// TwinCAT 3 PLC project PLC1
// ProgramVersion: 3.1.4023.0
// libraries:
//   CmpBitmapPool, * (System)
//   Tc2_MC2, * (Beckhoff Automation GmbH)
//   Tc2_Standard, * (Beckhoff Automation GmbH)
//   Tc2_System, * (Beckhoff Automation GmbH)
//   Tc3_Module, * (Beckhoff Automation GmbH)
//   VisuDialogs, * (System)
//   VisuSymbols,3.5.10.0,System
// project tree:
//   / GlobalTextList.TcGTLO (not stored), ImagePool.TcIPO (not stored), PlcTask.TcTTO, Visualization Manager.TcVMO (not stored)
//   GVLs/ GVL.TcGVL
//   POUs/ blinker.TcPOU (not stored), control.TcPOU, light.TcPOU, MAIN.TcPOU (not stored), motor.TcPOU
//   VISUs/ Huoltosivu.TcVIS (not stored), Visualization.TcVIS
// real-time tasks:
//   TASK PlcTask: cycle T#10ms, priority 20, ADS port 350
// motion (NC):
//   TASK NC-Task 1 SAF: cycle T#2ms, priority 4, ADS port 501
//   TASK NC-Task 1 SVB: cycle T#10ms, priority 8, ADS port 511
//   AXIS Axis 1, stepper (id 1)
//     Velo: Maximum=942.478
//     OtherSettings: AllowMotionCmdToSlave=true
//     encoder EncType=4
//       EncPara: ScaleFactorNumerator=0.007363107781851, MaxCount=#x0000ffff
//         Inc: RefSearchInverse=true, RefSyncInverse=false, RefMode=1, RefSoftSyncMask=#x0000ffff
//         TimeComp: TimeCompMode=1, EncDelayCycles=4
//     drive DrvType=24
//       Analog: VeloReferenz=942.477796076938, TorqueSetpointScale=10, ScaleFactorActTorque=0.1
//       TimeComp: TaskDelayCycles=1
//     controller CtrType=1
//       CtrPara: PriorControlFactor=1
//         Observer: BandWidth=20
//   AXIS Axis 2, servo (id 2)
//     OtherSettings: AllowMotionCmdToSlave=true
//     encoder EncType=19
//       EncPara: MaxCount=#xffffffff
//     drive DrvType=16
//       DrvPara: MaxCount=#xffffffff, DriveControlDWord=#x00020000
//         Analog: TorqueSetpointScale=10, ScaleFactorActTorque=0.1
//         TimeComp: TaskDelayCycles=1
//     controller CtrType=1
//       CtrPara: PriorControlFactor=1
//         Observer: BandWidth=20
// I/O:
//   DEVICE Device 1 (EtherCAT), AmsNetId 192.168.0.5.2.1
//     Term 1 (EK1200) [EK1200-5000 EtherCAT Power supply (2A E-Bus)]
//       Term 2 (EL1004) [EL1004 4Ch. Dig. Input 24V, 3ms]
//       Term 3 (EL1008) [EL1008 8Ch. Dig. Input 24V, 3ms]
//       Term 4 (EL2004) [EL2004 4Ch. Dig. Output 24V, 0.5A]
//       Term 5 (EL2008) [EL2008 8Ch. Dig. Output 24V, 0.5A]
//       Term 6 (EL3102) [EL3102 2Ch. Ana. Input +/-10V, Diff.]
//       Term 7 (EL4132) [EL4132 2Ch. Ana. Output +/-10V, 16bit]
//       Term 8 (EK1110) [EK1110 EtherCAT extension]
//     Term 9 (EK1100) [EK1100 EtherCAT Coupler (2A E-Bus)]
//       Term 10 (EL7031) [EL7031 1Ch. Stepper motor output stage (24V, 1.5A)]
//       Term 11 (EL7211-0010) [EL7211-0010 1Ch. MDP742 Servo motor output stage with OCT (50V, 4.5A RMS)]
//       Term 12 (EL9011) [EL9011 End Terminal]
//   DEVICE Device 5 (COM Port)
// variable links:
//   NC-Task 1 SAF/Axes/Axis 1, stepper <-> Device 1 (EtherCAT)/Term 9 (EK1100)/Term 10 (EL7031)
//     Drive/Inputs/In/nState1 @bit 3 <-> STM Status/Status/Error
//     Drive/Inputs/In/nState1 @bit 5 <-> STM Status/Status/Moving negative
//     Drive/Inputs/In/nState1 @bit 4 <-> STM Status/Status/Moving positive
//     Drive/Inputs/In/nState1 @bit 1 <-> STM Status/Status/Ready
//     Drive/Inputs/In/nState1 <-> STM Status/Status/Ready to enable
//     Drive/Inputs/In/nState1 @bit 6 <-> STM Status/Status/Torque reduced
//     Drive/Inputs/In/nState1 @bit 2 <-> STM Status/Status/Warning
//     Drive/Inputs/In/nState2 @bit 3 <-> STM Status/Status/Digital input 1
//     Drive/Inputs/In/nState2 @bit 4 <-> STM Status/Status/Digital input 2
//     Drive/Inputs/In/nState2 @bit 5 <-> STM Status/Status/Sync error
//     Drive/Inputs/In/nState2 @bit 7 <-> STM Status/Status/TxPDO Toggle
//     Drive/Inputs/In/nState4 @bit 1 <-> WcState/InputToggle
//     Drive/Inputs/In/nState4 <-> WcState/WcState
//     Drive/Outputs/Out/nCtrl1 <-> STM Control/Control/Enable
//     Drive/Outputs/Out/nCtrl1 @bit 2 <-> STM Control/Control/Reduce torque
//     Drive/Outputs/Out/nCtrl1 @bit 1 <-> STM Control/Control/Reset
//     Drive/Outputs/Out/nDataOut2[0] <-> STM Velocity/Velocity
//     Enc/Inputs/In/nDataIn1[0] <-> ENC Status compact/Counter value
//     Enc/Inputs/In/nDataIn2[0] <-> ENC Status compact/Latch value
//     Enc/Inputs/In/nState1 @bit 4 <-> ENC Status compact/Status/Counter overflow
//     Enc/Inputs/In/nState1 @bit 3 <-> ENC Status compact/Status/Counter underflow
//     Enc/Inputs/In/nState1 @bit 1 <-> ENC Status compact/Status/Latch extern valid
//     Enc/Inputs/In/nState1 @bit 2 <-> ENC Status compact/Status/Set counter done
//     Enc/Inputs/In/nState2 @bit 4 <-> ENC Status compact/Status/Status of extern latch
//     Enc/Inputs/In/nState2 @bit 5 <-> ENC Status compact/Status/Sync error
//     Enc/Inputs/In/nState2 @bit 7 <-> ENC Status compact/Status/TxPDO Toggle
//     Enc/Inputs/In/nState4 @bit 1 <-> WcState/InputToggle
//     Enc/Inputs/In/nState4 <-> WcState/WcState
//     Enc/Outputs/Out/nCtrl1 @bit 3 <-> ENC Control compact/Control/Enable latch extern on negative edge
//     Enc/Outputs/Out/nCtrl1 @bit 1 <-> ENC Control compact/Control/Enable latch extern on positive edge
//     Enc/Outputs/Out/nCtrl1 @bit 2 <-> ENC Control compact/Control/Set counter
//     Enc/Outputs/Out/nDataOut1[0] <-> ENC Control compact/Set counter value
//   NC-Task 1 SAF/Axes/Axis 2, servo <-> Device 1 (EtherCAT)/Term 9 (EK1100)/Term 11 (EL7211-0010)
//     Drive/Inputs/In/nDcOutputTime <-> InfoData/DcOutputShift
//     Drive/Inputs/In/nState1 <-> DRV Statusword/Statusword
//     Drive/Inputs/In/nState2 <-> DRV Statusword/Statusword @bit 8
//     Drive/Inputs/In/nState4 @bit 1 <-> WcState/InputToggle
//     Drive/Inputs/In/nState4 <-> WcState/WcState
//     Drive/Outputs/Out/nCtrl1 <-> DRV Controlword/Controlword
//     Drive/Outputs/Out/nCtrl2 <-> DRV Controlword/Controlword @bit 8
//     Drive/Outputs/Out/nDataOut2 <-> DRV Target velocity/Target velocity
//     Enc/Inputs/In/nDataIn1 <-> FB Position/Position
//     Enc/Inputs/In/nDcInputTime <-> InfoData/DcInputShift
//     Enc/Inputs/In/nState4 @bit 1 <-> WcState/InputToggle
//     Enc/Inputs/In/nState4 <-> WcState/WcState
//   PLC1/PLC1 Instance <-> Device 1 (EtherCAT)/Term 1 (EK1200)/Term 2 (EL1004)
//     PlcTask Inputs/GVL.safetyOk <-> Channel 1/GVL.safetyOk
//     PlcTask Inputs/motor.homingSensor <-> Channel 2/motor.homingSensor
//   PLC1/PLC1 Instance <-> Device 1 (EtherCAT)/Term 1 (EK1200)/Term 3 (EL1008)
//     PlcTask Inputs/GVL.playCCW <-> Channel 5/GVL.playCCW
//     PlcTask Inputs/GVL.playCW <-> Channel 4/GVL.playCW
//     PlcTask Inputs/GVL.reset <-> Channel 3/GVL.reset
//     PlcTask Inputs/GVL.start <-> Channel 6/GVL.start
//     PlcTask Inputs/GVL.stop <-> Channel 7/GVL.stop
//     PlcTask Inputs/GVL.tila1 <-> Channel 1/GVL.tila1
//     PlcTask Inputs/GVL.tila2 <-> Channel 2/GVL.tila2
//   PLC1/PLC1 Instance <-> Device 1 (EtherCAT)/Term 1 (EK1200)/Term 5 (EL2008)
//     PlcTask Outputs/GVL.playCCWBtnLight <-> Channel 3/GVL.playCCWBtnLight
//     PlcTask Outputs/GVL.resetBtnLight <-> Channel 1/GVL.resetBtnLight
//     PlcTask Outputs/GVL.safetyOkLight <-> Channel 4/GVL.safetyOkLight
//     PlcTask Outputs/GVL.stopBtnLight <-> Channel 5/GVL.stopBtnLight
//     PlcTask Outputs/GVL.systemOnLight <-> Channel 2/GVL.systemOnLight
//   PLC1/PLC1 Instance <-> Device 1 (EtherCAT)/Term 1 (EK1200)/Term 6 (EL3102)
//     PlcTask Inputs/GVL.potikka <-> AI Standard Channel 1/GVL.potikka
//   PLC1/PLC1 Instance <-> NC-Task 1 SAF/Axes/Axis 1, stepper
//     PlcTask Inputs/motor.stepperRef.NcToPlc <-> Outputs/ToPlc
//     PlcTask Outputs/motor.stepperRef.PlcToNc <-> Inputs/FromPlc

CONFIGURATION PLC1
    RESOURCE PLC ON TwinCAT3
        TASK PlcTask(INTERVAL := T#10ms, PRIORITY := 20);
        PROGRAM MAIN WITH PlcTask : MAIN;
    END_RESOURCE
END_CONFIGURATION

// ---- GVLs/GVL.TcGVL
{attribute 'qualified_only'}
VAR_GLOBAL
	
	//Laitteistoon liitetyt globaalit muuttujat:
	//Tulot:
	safetyOk AT%I*			: BOOL;
	start 	AT%I*			: BOOL;
	stop	AT%I*	 		: BOOL;
	playCW	AT%I*			: BOOL;
	playCCW	AT%I*			: BOOL;
	state1	AT%I*			: BOOL;
	state2	AT%I*			: BOOL;
	reset	AT%I*			: BOOL;
	potentioMeter AT%I*		: INT ;
	
	//GUI:
	
	startGUI 			: BOOL;
	stopGUI				: BOOL;
	resetGUI			: BOOL;
	positionResetGUI 	: BOOL;
	triggerGUI			: BOOL;

	//Lähdöt:

	systemOnLight		AT%Q*	: BOOL;
	safetyOkLight		AT%Q*	: BOOL;
	startBtnLight		AT%Q*	: BOOL;
	stopBtnLight		AT%Q*	: BOOL;
	resetBtnLight		AT%Q*	: BOOL;
	playCWBtnLight		AT%Q*	: BOOL;
	playCCWBtnLight		AT%Q*	: BOOL;
	
	//Muut globaalit muuttujat:
	
	driverMode		: INT := 0;
	errorMemory		: BOOL := TRUE;
	blinker1000ms	: BOOL;
	otherError		: BOOL;	
	systemOn		: BOOL;
	
END_VAR

// ---- POUs/control.TcPOU
PROGRAM control
VAR
	driverModeVar	: INT :=1;
	driverMode1		: BOOL;
	driverMode2		: BOOL;
	driverMode3		: BOOL;
	invisibleGUI	: BOOL := FALSE;
	visibleGUI		: BOOL := FALSE;
END_VAR

//Laitteen tilan asetus:
CASE GVL.driverMode OF
	1:	IF GVL.start AND NOT(GVL.errorMemory) THEN
			GVL.systemOn := TRUE;
			driverModeVar := GVL.driverMode;
		END_IF
		IF NOT(GVL.safetyOk) OR GVL.stop THEN
			GVL.systemOn := FALSE;
		END_IF
		
		IF NOT(GVL.safetyOk) THEN
			GVL.errorMemory := TRUE;
		END_IF
		IF GVL.reset THEN
			GVL.errorMemory := FALSE;
		END_IF
		
	2:	IF GVL.startGUI AND NOT(GVL.errorMemory) THEN
			GVL.systemOn := TRUE;
			driverModeVar := GVL.driverMode;
		END_IF
		IF NOT(GVL.safetyOk) OR GVL.stopGUI THEN
			GVL.systemOn := FALSE;
		END_IF
		
		IF NOT(GVL.safetyOk) THEN
			GVL.errorMemory := TRUE;
		END_IF
		IF GVL.resetGUI THEN
			GVL.errorMemory := FALSE;
		END_IF
		
	3:	IF GVL.startGUI AND NOT(GVL.errorMemory) THEN
			GVL.systemOn := TRUE;
			driverModeVar := GVL.driverMode;
		END_IF
		IF NOT(GVL.safetyOk) OR GVL.stopGUI THEN
			GVL.systemOn := FALSE;
		END_IF
		
		IF NOT(GVL.safetyOk) THEN
			GVL.errorMemory := TRUE;
		END_IF
		IF GVL.resetGUI THEN
			GVL.errorMemory := FALSE;
		END_IF
		
END_CASE

IF driverModeVar <> GVL.driverMode THEN
	GVL.systemOn := FALSE;
END_IF

IF GVL.driverMode = 3 THEN
	invisibleGUI := TRUE;
	visibleGUI := FALSE;
ELSE
	invisibleGUI := FALSE;
	visibleGUI := TRUE; 
END_IF

//IF GVL.start THEN
//	driverModeVar := GVL.driverMode;
//END_IF

IF GVL.state1 AND NOT(GVL.state2) THEN
	GVL.driverMode := 1;
	driverMode1 := FALSE;
ELSE
	driverMode1 := TRUE;
END_IF

IF NOT(GVL.state2) AND NOT(GVL.state1) THEN
	GVL.driverMode := 2;
	driverMode2 := FALSE;
ELSE
	driverMode2 := TRUE;
END_IF

IF NOT(GVL.state1) AND GVL.state2 THEN
	GVL.driverMode := 3;
	driverMode3 := FALSE;
ELSE
	driverMode3 := TRUE;
END_IF

END_PROGRAM

// ---- POUs/light.TcPOU
PROGRAM light
VAR
	otherError	: BOOL;
END_VAR


IF GVL.systemOn OR GVL.playCW THEN
	GVL.systemOnLight := TRUE;
ELSIF (NOT(GVL.errorMemory) AND GVL.blinker1000ms) THEN
	GVL.systemOnLight := TRUE;
ELSE
	GVL.systemOnLight :=FALSE;
END_IF

IF GVL.stop THEN
	GVL.stopBtnLight := TRUE;
ELSE
	GVL.stopBtnLight :=FALSE;
END_IF

IF GVL.playCCW THEN
	GVL.playCCWBtnLight := TRUE;
ELSE
	GVL.playCCWBtnLight :=FALSE;
END_IF

IF NOT(GVL.safetyOk) OR GVL.start THEN
	GVL.safetyOkLight := TRUE;
ELSE
	IF  GVL.blinker1000ms AND (otherError OR GVL.errorMemory) THEN
		GVL.safetyOkLight := TRUE;
	ELSE
		GVL.safetyOkLight := FALSE;
	END_IF
	
	IF GVL.errorMemory AND NOT(otherError) OR gvl.reset THEN
		GVL.resetBtnLight := TRUE;	
	ELSE
		GVL.resetBtnLight := FALSE;
	END_IF
END_IF

END_PROGRAM

// ---- POUs/motor.TcPOU
PROGRAM motor
VAR
	stepperRef				: AXIS_REF;
	stepperPower			: MC_Power;
	stepperMoveAbsolute		: MC_MoveAbsolute;
	JOG						: MC_jog;
	Homing					: MC_Home; //usermode 3 varten
	stepperReset			: MC_reset;
	
	stepperValue			: INT := 0;
	stepperSpeed			: INT := 100;
	stepperSpeedGUI			: INT := 0;
	stepperSpeedVay			: INT := 0;
	stepperValueVay			: INT := 0;
	currentStepperSpeed		: LREAL;
	currentStepperPosition	: LREAL;
	arvo					: INT;
	homingSensor AT%I*		: BOOL;
	
	calibrationBtn			: BOOL;
	approachSensor			: BOOL;
	inReference				: BOOL;
	positionMatch			: BOOL;
	inReferenceVar			: BOOL;
	
END_VAR

stepperPower(
	Axis:= stepperRef, 
	Enable:= , 
	Enable_Positive:= TRUE, 
	Enable_Negative:= TRUE, 
	Override:= stepperSpeed, 
	BufferMode:= , 
	Options:= , 
	Status=> , 
	Busy=> , 
	Active=> , 
	Error=> , 
	ErrorID=> );
	
stepperMoveAbsolute(
	Axis:= stepperRef, 
	Execute:= , 
	Position:= , 
	Velocity:= , 
	Acceleration:= , 
	Deceleration:= , 
	Jerk:= , 
	BufferMode:= , 
	Options:= , 
	Done=> , 
	Busy=> , 
	Active=> , 
	CommandAborted=> , 
	Error=> , 
	ErrorID=> );
	
JOG(
	Axis:= stepperRef, 
	JogForward:= , 
	JogBackwards:= , 
	Mode:= , 
	Position:= , 
	Velocity:= , 
	Acceleration:= , 
	Deceleration:= , 
	Jerk:= , 
	Done=> , 
	Busy=> , 
	Active=> , 
	CommandAborted=> , 
	Error=> , 
	ErrorID=> );	

Homing(
	Axis:= stepperRef, 
	Execute:= , 
	Position:= , 
	HomingMode:= , 
	BufferMode:= , 
	Options:= , 
	bCalibrationCam:= , 
	Done=> , 
	Busy=> , 
	Active=> , 
	CommandAborted=> , 
	Error=> , 
	ErrorID=> );

stepperReset(
	Axis:= stepperRef, 
	Execute:= , 
	Done=> , 
	Busy=> , 
	Error=> , 
	ErrorID=> );
	

IF GVL.systemOn THEN
	stepperPower.Enable	:= TRUE;
	
	CASE GVL.driverMode OF
		
		1:	positionMatch	:= FALSE;
			inReference		:= FALSE;
		
			IF GVL.playCCW THEN
				JOG.JogForward := TRUE;
			ELSE
				JOG.JogForward := FALSE;
			END_IF
				
			IF GVL.playCW THEN
				JOG.JogBackwards := TRUE;
			ELSE
				JOG.JogBackwards := FALSE;
			END_IF
			
			arvo 					:=	(gvl.potentioMeter / 325);
			stepperSpeed			:= arvo;
			stepperPower.Override	:= stepperSpeed;	
				
		2:	homing.HomingMode		:= MC_Direct;
			positionMatch			:= FALSE;
			inReference				:= FALSE;
			
			IF GVL.positionResetGUI THEN
				homing.Execute			:= TRUE;
				homing.Position			:= 0;
				currentStepperPosition	:= 0;
			ELSE
				homing.Execute := FALSE;
			END_IF
				
			IF GVL.triggerGUI THEN
				stepperMoveAbsolute.Position	:= stepperValue;
				stepperMoveAbsolute.Velocity 	:= stepperSpeedGUI;
				//stepperPower.Override			:= stepperSpeedGUI;
				stepperMoveAbsolute.Execute		:= TRUE;
			END_IF
				
			IF stepperMoveAbsolute.Done THEN
				stepperMoveAbsolute.Execute 	:= FALSE;
			END_IF
				
		3:	homing.HomingMode	:= MC_DefaultHoming;
		
			IF calibrationBtn THEN
				homing.Execute			:= TRUE;
				positionMatch			:= FALSE;
			ELSE
				homing.Execute			:= FALSE;
				homing.bCalibrationCam	:= FALSE;	
			END_IF
			
			IF homingSensor THEN
				homing.bCalibrationCam	:= TRUE;
				inReference				:= TRUE;
				inReferenceVar			:= TRUE;
				homing.Execute			:= FALSE;
			END_IF
						
			IF inReference THEN
				homing.Position			:= 0;
				currentStepperPosition	:= 0;
				IF GVL.triggerGUI THEN
					stepperMoveAbsolute.Position	:= stepperValueVay;
					stepperMoveAbsolute.Velocity 	:= stepperSpeedVay;
					//stepperPower.Override			:= stepperSpeedVay;
					stepperMoveAbsolute.Execute		:= TRUE;
					inReferenceVar					:= FALSE;
					positionMatch					:= FALSE;
				END_IF
			END_IF
			
			IF stepperMoveAbsolute.Done THEN
				positionMatch					:= TRUE;
				stepperMoveAbsolute.Execute 	:= FALSE;
			END_IF		
								
	END_CASE
	currentStepperSpeed 			:= stepperRef.NcToPlc.ActVelo;
	currentStepperPosition			:= stepperRef.NcToPlc.ActPos;
ELSE
	stepperPower.Enable			:= FALSE;
	stepperMoveAbsolute.Execute	:= FALSE;
	homing.Execute				:= FALSE;
END_IF

IF GVL.reset OR gvl.resetGUI OR GVL.start OR gvl.startGUI THEN
	stepperReset.Execute	:= TRUE;
ELSE
	stepperReset.Execute	:= FALSE;
END_IF

END_PROGRAM

// ---- VISUs/Visualization.TcVIS
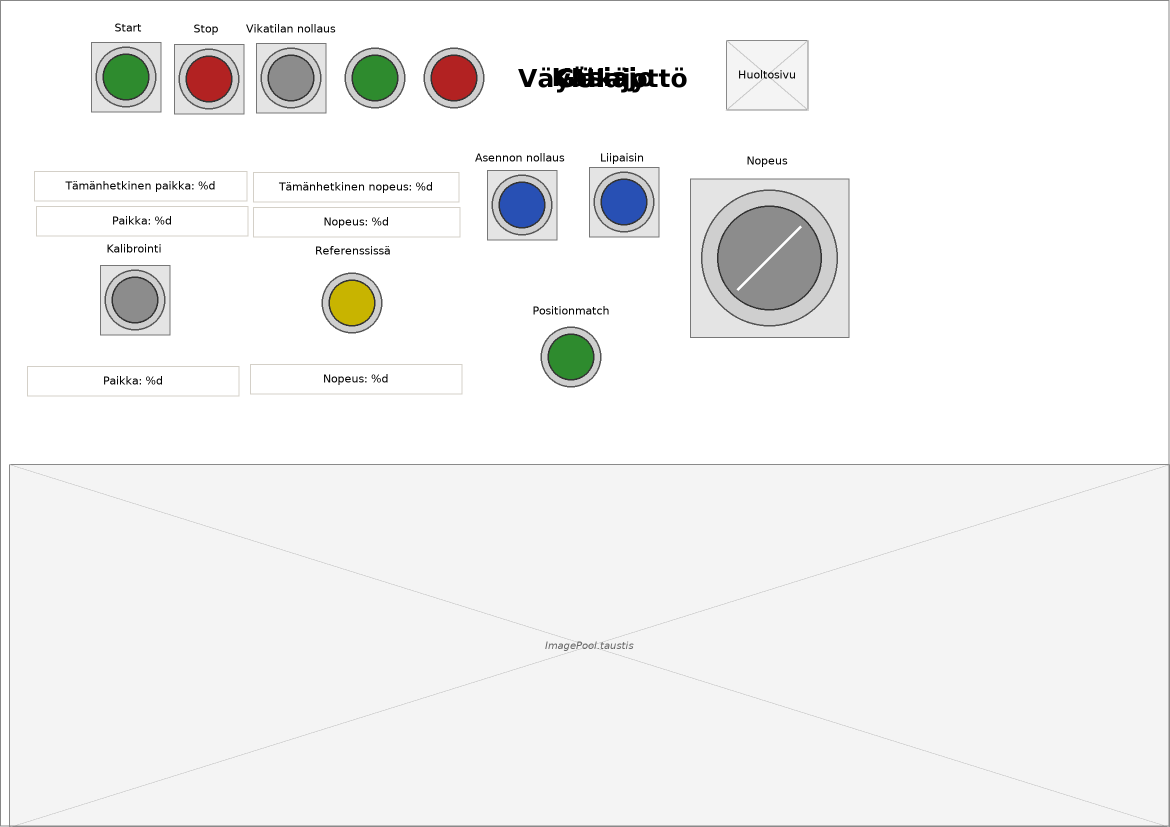
VISUALIZATION Visualization  // 1170x827, background image ImagePool.taustis2
    PushSwitch (91,42 70x70), variable: GVL.startGUI, behaviour: TAP, style: Switch-PushSwitch-Green
    PushSwitch (174,44 70x70), variable: GVL.stopGUI, behaviour: TAP, style: Switch-PushSwitch-Red
    PushSwitch (256,43 70x70), variable: GVL.resetGUI, behaviour: TAP, style: Switch-PushSwitch-Gray
    Lamp1 (340,43 70x70), variable: GVL.systemOnLight, style: Lamp-Lamp1-Green
    Label (526,63 150x30), "GUIajo", invisible if: control.driverMode2
    Label (528,62 150x30), "Käsiajo", invisible if: control.driverMode1
    Label (503,63 200x30), "Väyläkäyttö", invisible if: control.driverMode3
    Lamp1 (419,43 70x70), variable: GVL.safetyOkLight, style: Lamp-Lamp1-Red
    Textfield (36,206 212x30), "Paikka: %d", text variable: motor.stepperValue, invisible if: control.invisibleGUI
        OnMouseDown: write the text variable via Default
    Textfield (253,207 207x30), "Nopeus: %d", text variable: motor.stepperSpeedGUI, invisible if: control.invisibleGUI
    Textfield (34,171 213x30), "Tämänhetkinen paikka: %d", text variable: motor.currentStepperPosition
    Textfield (253,172 206x30), "Tämänhetkinen nopeus: %d", text variable: motor.CurrentStepperSpeed
    PushSwitch (487,170 70x70), variable: GVL.asemannollausGUI, invisible if: control.invisibleGUI, behaviour: TAP, style: Switch-PushSwitch-Blue
    Label (445,143 150x30), "Asennon nollaus", invisible if: control.invisibleGUI
    Label (216,14 150x30), "Vikatilan nollaus"
    Label (131,14 150x30), "Stop"
    Label (53,13 150x30), "Start"
    PushSwitch (589,167 70x70), variable: GVL.triggerGUI, behaviour: TAP, style: Switch-PushSwitch-Blue
    Label (547,143 150x30), "Liipaisin"
    PushSwitch (100,265 70x70), variable: motor.kalibrointibtn, invisible if: control.visibleGUI, behaviour: TAP, style: Switch-PushSwitch-Gray
    Image (9,464 1161x363), image: ImagePool.taustis
    Label (59,234 150x30), "Kalibrointi", invisible if: control.visibleGUI
    Lamp1 (317,268 70x70), variable: motor.referenssissaVar, invisible if: control.visibleGUI, style: Lamp-Lamp1-Yellow
    Label (278,236 150x30), "Referenssissä", invisible if: control.visibleGUI
    Label (692,146 150x30), "Nopeus", invisible if: control.invisibleGUI
    Image (726,40 82x70), "Huoltosivu", image: VisuDialogs.ImagePoolDialogs.FileOpen
        OnMouseClick: change screen: Huoltosivu
    Textfield (250,364 212x30), "Nopeus: %d", text variable: motor.stepperSpeedVay, invisible if: control.visibleGUI
        OnMouseDown: write the text variable via Default
    Textfield (27,366 212x30), "Paikka: %d", text variable: motor.stepperValueVay, invisible if: control.visibleGUI
        OnMouseDown: write the text variable via Default
    Potentiometer360 (690,177 159x162), variable: motor.stepperSpeedGUI, style: Potentiometer-Potentiometer360-Gray, scale format: %.1f, scale 0..100
        p2431819421: Outside
    Lamp1 (536,322 70x70), variable: motor.positionMatch, invisible if: control.visibleGUI, style: Lamp-Lamp1-Green
    Label (496,296 150x30), "Positionmatch", invisible if: control.visibleGUI
END_VISUALIZATION
